INTERFACE I_HostMetadata EXTENDS __SYSTEM.IQueryInterface

PROPERTY Metadatum : I_Metadatum
GET
END_GET
END_PROPERTY

END_INTERFACE

(* stored: Version 1.1.0.1, ProductVersion 3.1.4024.12
   Itf I_HostMetadata: Id {de299323-ae26-4fca-8708-1ea7c86e8f21}
   Property Metadatum: Id {ff3ce6a8-7126-4425-9724-441dfcb735fd}
   Get Get: Id {17482e91-f039-4e0b-84e5-7f5e9ec0fc0a} *)
